// TwinCAT 3 PLC project PLC_PML
// ProgramVersion: 3.1.4023.0
// libraries:
//   PML_Base_Library, * (SPT)
//   Tc2_Math, * (Beckhoff Automation GmbH)
//   Tc2_MC2, * (Beckhoff Automation GmbH)
//   Tc2_MC2_Drive, * (Beckhoff Automation GmbH)
//   Tc2_Standard, * (Beckhoff Automation GmbH)
//   Tc2_System, * (Beckhoff Automation GmbH)
//   Tc2_Utilities, * (Beckhoff Automation GmbH)
//   Tc3_EventLogger, * (Beckhoff Automation GmbH)
//   Tc3_Module, * (Beckhoff Automation GmbH)
//   Tc3_PackML_V2, * (Beckhoff Automation GmbH)
// project tree:
//   Application/01_Application_Level_Items/02_DUT/01_ENUM/ E_PMLUnitMode.TcDUT
//   Application/01_Application_Level_Items/02_DUT/02_STRUCT/ ST_ProductionData_HMI.TcDUT
//   Application/01_Application_Level_Items/02_DUT/03_ALIAS/ T_PackMLTags.TcDUT
//   Application/01_Application_Level_Items/03_ITFs/ ITF_ProductionData.TcIO
//   Application/01_Application_Level_Items/04_HMI_Connections/ FB_MainModule_HMI_Connection.TcPOU, ST_PMLControl.TcDUT, ST_PMLControl_Simplified.TcDUT
//   Application/01_Application_Level_Items/999_VISU/ V_Application.TcVIS (not stored)
//   Application/01_Application_Level_Items/99_Templates/ FB_Module_TEMPLATE.TcPOU
//   Application/01_Application_Level_Items/ FB_ProductionMonitor.TcPOU
//   Application/02_MachineModules/ FB_TestMachine.TcPOU
//   Application/03_EquipmentModules/ FB_TestEquipment.TcPOU
//   Application/04_Components/01_Cylinder_Example/ FB_CylinderBase.TcPOU, ITF_CylinderBase.TcIO, ST_CylinderBase_HMI.TcDUT
//   Application/ MAIN.TcPOU
//   / GlobalTextList.TcGTLO (not stored), PlcTask.TcTTO (not stored), Visualization Manager.TcVMO (not stored)
// real-time tasks:
//   TASK PlcTask: cycle T#1ms, priority 20, ADS port 350
//   TASK VISU_TASK: cycle T#200000us, priority 30, ADS port 351
//   TASK Job Task: cycle default, priority 32
//   TASK MC-Task (MET): cycle T#2ms, priority 3, ADS port 521
//   TASK MC-Task (MPT): cycle T#10ms, priority 8, ADS port 531
// motion (NC):
//   TASK NC-Task 1 SAF: cycle T#2ms, priority 4, ADS port 501
//   TASK NC-Task 1 SVB: cycle T#10ms, priority 9, ADS port 511
//   AXIS Axis 1 (id 1)
//     General: UnitFlags=#x00000004
//     Dynamic: AccelerationMaximum=10000, DecelerationMaximum=10000, Acceleration=1000, Deceleration=1000, Jerk=1750
//     Velo: Maximum=1500
//     OtherSettings: AllowMotionCmdToSlave=true
//     encoder EncType=1
//       EncPara: ModuloFactor=720
//     drive DrvType=5
//       Analog: TorqueSetpointScale=10, ScaleFactorActTorque=0.1
//       TimeComp: TaskDelayCycles=1
//     controller CtrType=1
//       CtrPara: PriorControlFactor=1
//         Observer: BandWidth=20
//   AXIS Axis 2 (id 2)
//     General: UnitFlags=#x00000004
//     OtherSettings: AllowMotionCmdToSlave=true
//     encoder EncType=1
//     drive DrvType=5
//       Analog: TorqueSetpointScale=10, ScaleFactorActTorque=0.1
//       TimeComp: TaskDelayCycles=1
//     controller CtrType=1
//       CtrPara: PriorControlFactor=1
//         Observer: BandWidth=20

// ---- Application/01_Application_Level_Items/02_DUT/01_ENUM/E_PMLUnitMode.TcDUT
{attribute 'qualified_only'} //Note that this is not "Strict" since it needs to interact with the mode manager, which uses DINTs for mode
TYPE E_PMLUnitMode : (
        ePMLUnitMode_Invalid     := 0,
        ePMLUnitMode_Production  := 1,
        ePMLUnitMode_Maintenance := 2,
        ePMLUnitMode_Manual      := 3
    // User defined modes
    (*ePMLUnitMode_SemiAutomatic  :=  4,
    ePMLUnitMode_DryRun         :=  5,
	ePMLUnitMode_Standalone		:=  6,
	ePMLUnitMode_Usermode4		:=  7,
	ePMLUnitMode_Usermode5 		:=  8,
	ePMLUnitMode_Usermode6 		:=  9,
	ePMLUnitMode_Usermode7 		:=  10 *)
    ) DINT;
END_TYPE

// ---- Application/01_Application_Level_Items/02_DUT/02_STRUCT/ST_ProductionData_HMI.TcDUT
TYPE ST_ProductionData_HMI :
    STRUCT
        bHMIControlAvailable    : BOOL; //Set TRUE *FROM PLC* when HMI requests can be processed
        bIncomingHMIRequest     : BOOL; //Pulses TRUE when an HMI request is issued
        bHMICommandConfirmation : BOOL; //Confirms receipt and subsequent processing of the command sent by the HMI

        bShiftLengthHMISetRequest : BOOL;
        tShiftLengthHMISetValue   : TIME;

        bShiftProductionTargetHMISetRequest : BOOL;
        nShiftProductionTargetHMISetValue   : DINT;

        bWarningMarginHMISetRequest : BOOL;
        fWarningMarginHMISetValue   : LREAL;

        bProductionRateHMISetRequest : BOOL;
        fProductionRateHMISetValue   : LREAL;

        tShiftLength           : TIME; //Specify the time duration of a shift
        nShiftProductionTarget : DINT; //Specify the desired production count by end of shift

        nCurrentAcceptableProductionCount : DINT;
        nCurrentWarningProductionCount    : DINT;
        nCurrentShiftProductionCount      : DINT; //Number of products completed so far on the current shift
        nCurrentShiftTarget               : DINT; //Expected number of completed products at the current time in the shift
        tCurrentShiftTime                 : TIME; //Time elapsed since the start of the shift
        tRemainingShiftTime               : TIME; //Time remaining in the current shift
        tShiftStartTimeStamp              : TIMESTRUCT;
        tShiftStartTimeStamp_UTC          : STRING;
        fProductionRate_Setpoint          : LREAL;
        fProductionRate_Actual            : LREAL;
        fProductionRate_Required          : LREAL;

    END_STRUCT
END_TYPE

// ---- Application/01_Application_Level_Items/02_DUT/03_ALIAS/T_PackMLTags.TcDUT
(*	Change the type depending on the needs, minimum packml set or full
Tc3_PackML_V2.ST_PackMLv30 // Tc3_PackML_V2.ST_PackMLv30min*)
TYPE T_PackMLTags : Tc3_PackML_V2.ST_PackMLv30;
END_TYPE

// ---- Application/01_Application_Level_Items/04_HMI_Connections/ST_PMLControl.TcDUT
TYPE ST_PMLControl :
    STRUCT
        bNewCommand   : BOOL;
        bConfirmation : BOOL;

        eMode        : E_PMLUnitMode;
        eModeCommand : E_PMLUnitMode;

        eState        : E_PMLState;
        eStateCommand : E_PMLCommand;

        a_sModeNames : ARRAY[0..31] OF STRING;
    END_STRUCT
END_TYPE

// ---- Application/01_Application_Level_Items/04_HMI_Connections/ST_PMLControl_Simplified.TcDUT
TYPE ST_PMLControl_Simplified :
    STRUCT
        bConfirmation : BOOL;

        bClearEnabled : BOOL;
        bResetEnabled : BOOL;
        bStartEnabled : BOOL;
        bStopEnabled  : BOOL;

        bClearPressed : BOOL;
        bResetPressed : BOOL;
        bStartPressed : BOOL;
        bStopPressed  : BOOL;
    END_STRUCT
END_TYPE

// ---- Application/04_Components/01_Cylinder_Example/ST_CylinderBase_HMI.TcDUT
TYPE ST_CylinderBase_HMI :
    STRUCT
        //Status information
        tExtendTime     : TIME;
        tRetractTime    : TIME;
        fTimeoutFactor  : LREAL;
        bExtended       : BOOL;
        bRetracted      : BOOL;
        bExtending      : BOOL;
        bRetracting     : BOOL;
        bRetractCommand : BOOL;
        bExtendCommand  : BOOL;

        //Control information
        bHMIControlAvailable    : BOOL; //Set TRUE *FROM PLC* when HMI requests can be processed
        bIncomingHMIRequest     : BOOL; //Pulses TRUE when an HMI request is issued
        bHMICommandConfirmation : BOOL; //Confirms receipt and subsequent processing of the command sent by the HMI

        bExtendHMIRequest           : BOOL;  //HMI requests to extend the cylinder
        bRetractHMIRequest          : BOOL;  //HMI requests to retract the cylinder
        bIdleHMIRequest             : BOOL;  //HMI requests to idle the cylinder (no active output)
        bExtendTimeHMISetRequest    : BOOL;  //HMI requests to set the cylinder's expected extend time
        tExtendTimeHMISetValue      : TIME;  //HMI setpoint value for the expected extend time
        bRetractTimeHMISetRequest   : BOOL;  //HMI requests to set the cylinder's expected retract time
        tRetractTimeHMISetValue     : TIME;  //HMI setpoint value for the expected retract time
        bTimeoutFactorHMISetRequest : BOOL;  //HMI requests to set the timeout factor for the cylinder
        fTimeoutFactorHMISetValue   : LREAL; //HMI setpoint value for the cylinder's timeout factor
    END_STRUCT
END_TYPE

// ---- Application/01_Application_Level_Items/03_ITFs/ITF_ProductionData.TcIO
INTERFACE ITF_ProductionData

PROPERTY CurrentShiftAcceptableProduction : DINT
GET
END_GET
SET
END_SET
END_PROPERTY

PROPERTY CurrentShiftProductionCount : DINT
GET
END_GET
END_PROPERTY

PROPERTY CurrentShiftTarget : DINT
GET
END_GET
END_PROPERTY

PROPERTY CurrentShiftTime : TIME
GET
END_GET
END_PROPERTY

PROPERTY CurrentShiftWarningProduction : DINT
GET
END_GET
SET
END_SET
END_PROPERTY

PROPERTY NewProductionRate : bool
GET
END_GET
END_PROPERTY

PROPERTY ProductComplete : bool
GET
END_GET
SET
END_SET
END_PROPERTY

PROPERTY ProductionRate_Actual : lreal
GET
END_GET
END_PROPERTY

PROPERTY ProductionRate_Required : lreal
GET
END_GET
SET
END_SET
END_PROPERTY

PROPERTY ProductionRate_Setpoint : lreal
GET
END_GET
SET
END_SET
END_PROPERTY

PROPERTY RateAveragingCount : DINT
GET
END_GET
SET
END_SET
END_PROPERTY

PROPERTY RemainingShiftTime : TIME
GET
END_GET
SET
END_SET
END_PROPERTY

PROPERTY ShiftComplete : BOOL
GET
END_GET
END_PROPERTY

PROPERTY ShiftLength : TIME
GET
END_GET
SET
END_SET
END_PROPERTY

PROPERTY ShiftProductionTarget : DINT
GET
END_GET
SET
END_SET
END_PROPERTY

PROPERTY WarningMargin : LREAL //0 to 100, interpreted as a percentage difference between the current rate and the required rate to meet the production target, decimal values permitted
GET
END_GET
SET
END_SET
END_PROPERTY

END_INTERFACE

// ---- Application/04_Components/01_Cylinder_Example/ITF_CylinderBase.TcIO
INTERFACE ITF_CylinderBase //cylinder no feedback spring return solonoid

METHOD Extend : BOOL
END_METHOD

PROPERTY Extended : BOOL //Status bit for the position of the cylinder
GET
END_GET
END_PROPERTY

PROPERTY Extending : BOOL
GET
END_GET
END_PROPERTY

PROPERTY ExtendTime : TIME //Approximate expected time for the cylinder to complete an extension cycle
GET
END_GET
SET
END_SET
END_PROPERTY

METHOD Idle : BOOL
END_METHOD

METHOD Retract : UDINT
END_METHOD

PROPERTY Retracted : BOOL //Status bit for the position of the cylinder
GET
END_GET
END_PROPERTY

PROPERTY Retracting : BOOL
GET
END_GET
END_PROPERTY

PROPERTY RetractTime : TIME
GET
END_GET
SET
END_SET
END_PROPERTY

PROPERTY TimeoutFactor : LREAL //Multiplicative factor that determines error timeout threshold based on the expected time
GET
END_GET
SET
END_SET
END_PROPERTY

END_INTERFACE

// ---- Application/01_Application_Level_Items/04_HMI_Connections/FB_MainModule_HMI_Connection.TcPOU
FUNCTION_BLOCK FB_MainModule_HMI_Connection
VAR CONSTANT
    //Constant declarations
    PRODUCTION_DATA_ALARM_COUNT : UDINT := 16;
END_VAR
VAR PERSISTENT
    //ITF_ProductionData internal variables
    tShiftLength             : TIME  := T#10M;
    nShiftProductionTarget   : DINT  := 1000;
    fWarningMargin           : LREAL := 10;
    fProductionRate_Setpoint : LREAL := 30;
    nRateAveragingCount      : DINT  := 10;
END_VAR
VAR
    //Internal Property Variables
    itfMainModule : ITF_PMLModuleBase;

    //Program Tree variables
    fbModuleTree         : FB_Tree_IndexBased;
    a_stMachineTreeNodes : ARRAY[0..63] OF ST_Tree_IndexBased_Node;
    sTopLevelMachine     : STRING;

    //PML Control Variables
    stMainPMLControl_Simplified : ST_PMLControl_Simplified;
    stMainPMLControl_Standard   : ST_PMLControl;

    //Status Variables
    stMainProductionData : REFERENCE TO ST_ProductionData_HMI;

    //Production Data variables
    bShiftComplete                    : BOOL;
    bProductComplete                  : BOOL;
    nCurrentShiftProductionCount      : INT;
    nCurrentShiftTarget               : DINT;
    tCurrentShiftTime                 : TIME;
    tRemainingShiftTime               : TIME;
    tShiftStartTimeStamp              : TIMESTRUCT;
    tShiftStartTimeStamp_UTC          : STRING;
    nCurrentWarningProductionCount    : DINT;
    nCurrentAcceptableProductionCount : DINT;

    fProductionRate_Required : LREAL;
    fProductionRate_Actual   : LREAL;

    a_nLastProductTimestamps : ARRAY[1..100] OF ULINT; //Array of ULINT values (1 unit = 1ns) for the relative time of each of the last 100 completed products
    fbShiftTimer             : TON;
    fbGetTime                : NT_GetTime;
    fbProductComplete_RT     : R_TRIG;

    bResetMaxProductionCount   : BOOL;
    bResetTotalProductionCount : BOOL;

    nMaxProductionCount   : DINT;
    nTotalProductionCount : DINT;

    stProductionDataHMI      : ST_ProductionData_HMI;
    fbFIFO                   : FB_FIFO_ULINT_Array;
    a_fbProductionDataAlarms : ARRAY[1..PRODUCTION_DATA_ALARM_COUNT] OF FB_TcAlarm;
    fTemp                    : LREAL;

    //Other Internal Variables
    bInitialized : BOOL;
    i            : UDINT;

END_VAR

METHOD CyclicLogic : BOOL
VAR_INPUT
END_VAR
IF NOT bInitialized THEN
    initialize();
    bInitialized := TRUE;
END_IF

stMainPMLControl_Standard.eMode  := itfMainModule.Mode;
stMainPMLControl_Standard.eState := itfMainModule.State;

FOR i := 1 TO 5 DO
    stMainPMLControl_Standard.a_sModeNames[i] := F_UnitModeToString(i);
	
END_FOR

stMainPMLControl_Standard.eState := itfMainModule.State;
stMainPMLControl_Standard.eMode  := itfMainModule.Mode;

MainCycleControl();

//bProductComplete := itfMainModule.ProductComplete;

ProductionMonitor();
HMICommunication();

//itfMainModule.ProductionRate_Setpoint := fProductionRate_Setpoint;
END_METHOD

PROPERTY DataStructure_Adder : ITF_Tree_IndexBased
GET
DataStructure_Adder := fbModuleTree;
END_GET
END_PROPERTY

METHOD HMICommunication : BOOL
VAR_INPUT
END_VAR
//Production Data================================================================================================================================================

//Process HMI requests
IF stProductionDataHMI.bIncomingHMIRequest AND NOT stProductionDataHMI.bHMICommandConfirmation
    THEN //If a request has been issued by the HMI, and a previous request has not just E_SequenceState.Finished being processed
    IF stProductionDataHMI.bShiftProductionTargetHMISetRequest THEN
        nShiftProductionTarget                      := stProductionDataHMI.nShiftProductionTargetHMISetValue;
        stProductionDataHMI.bHMICommandConfirmation := TRUE; //Confirm that the request has been processed
    END_IF

    IF stProductionDataHMI.bWarningMarginHMISetRequest THEN
        fWarningMargin                              := stProductionDataHMI.fWarningMarginHMISetValue;
        stProductionDataHMI.bHMICommandConfirmation := TRUE; //Confirm that the request has been processed
    END_IF

    IF stProductionDataHMI.bShiftLengthHMISetRequest THEN
        tShiftLength                                := stProductionDataHMI.tShiftLengthHMISetValue;
        stProductionDataHMI.bHMICommandConfirmation := TRUE; //Confirm that the request has been processed
    END_IF

    IF stProductionDataHMI.bProductionRateHMISetRequest THEN
        fProductionRate_Setpoint                    := stProductionDataHMI.fProductionRateHMISetValue;
        stProductionDataHMI.bHMICommandConfirmation := TRUE; //Confirm that the request has been processed
    END_IF
END_IF

//Update HMI Status Info
stProductionDataHMI.tShiftLength                      := tShiftLength;
stProductionDataHMI.nShiftProductionTarget            := nShiftProductionTarget;
stProductionDataHMI.nCurrentShiftProductionCount      := nCurrentShiftProductionCount;
stProductionDataHMI.nCurrentShiftTarget               := nCurrentShiftTarget;
stProductionDataHMI.nCurrentAcceptableProductionCount := nCurrentAcceptableProductionCount;
stProductionDataHMI.nCurrentWarningProductionCount    := nCurrentWarningProductionCount;
stProductionDataHMI.tCurrentShiftTime                 := tCurrentShiftTime;
stProductionDataHMI.tRemainingShiftTime               := tRemainingShiftTime;
stProductionDataHMI.tShiftStartTimeStamp              := tShiftStartTimeStamp;
stProductionDataHMI.tShiftStartTimeStamp_UTC          := tShiftStartTimeStamp_UTC;
stProductionDataHMI.fProductionRate_Setpoint          := F_LREAL_RoundToPlace(fProductionRate_Setpoint, 1);
stProductionDataHMI.fProductionRate_Actual            := F_LREAL_RoundToPlace(fProductionRate_Actual, 1);
stProductionDataHMI.fProductionRate_Required          := F_LREAL_RoundToPlace(fProductionRate_Required, 1);
END_METHOD

METHOD initialize : BOOL
VAR_INPUT
END_VAR
sTopLevelMachine := itfMainModule.ModuleName;

fbModuleTree(a_stNodes := a_stMachineTreeNodes, sHead := sTopLevelMachine);

F_CreateAllEventsInClass(p_aAlarms  := a_fbProductionDataAlarms,
                         nClassSize := SIZEOF(TC_EVENTS.ProductionData),
                         pInitEvent := ADR(TC_EVENTS.ProductionData.InitReferenceEvent),
                         sPrefix    := MainModule.ModuleName);
END_METHOD

METHOD MainCycleControl : BOOL
VAR_INPUT
END_VAR
//Simplified Commands
//Handle button presses
IF NOT stMainPMLControl_Simplified.bConfirmation AND stMainPMLControl_Simplified.bStartPressed THEN
    IF stMainPMLControl_Standard.eState = Tc3_PackML_V2.E_PMLState.ePMLState_Idle THEN
        itfMainModule.StateCommand := Tc3_PackML_V2.E_PMLCommand.ePMLCommand_Start;
    ELSIF stMainPMLControl_Standard.eState = Tc3_PackML_V2.E_PMLState.ePMLState_Held THEN
        itfMainModule.StateCommand := Tc3_PackML_V2.E_PMLCommand.ePMLCommand_Unhold;
    END_IF

    stMainPMLControl_Simplified.bConfirmation := TRUE;
END_IF

IF NOT stMainPMLControl_Simplified.bConfirmation AND stMainPMLControl_Simplified.bStopPressed THEN
    itfMainModule.StateCommand                := Tc3_PackML_V2.E_PMLCommand.ePMLCommand_Stop;
    stMainPMLControl_Simplified.bConfirmation := TRUE;
END_IF

IF NOT stMainPMLControl_Simplified.bConfirmation AND stMainPMLControl_Simplified.bResetPressed THEN
    itfMainModule.StateCommand                := Tc3_PackML_V2.E_PMLCommand.ePMLCommand_Reset;
    stMainPMLControl_Simplified.bConfirmation := TRUE;
END_IF

IF NOT stMainPMLControl_Simplified.bConfirmation AND stMainPMLControl_Simplified.bClearPressed THEN
    itfMainModule.StateCommand                := Tc3_PackML_V2.E_PMLCommand.ePMLCommand_Clear;
    stMainPMLControl_Simplified.bConfirmation := TRUE;
END_IF

//Handle enabling of the Start button
IF stMainPMLControl_Standard.eState = Tc3_PackML_V2.E_PMLState.ePMLState_Idle
       OR stMainPMLControl_Standard.eState = Tc3_PackML_V2.E_PMLState.ePMLState_Held THEN
    stMainPMLControl_Simplified.bStartEnabled := TRUE;
ELSE
    stMainPMLControl_Simplified.bStartEnabled := FALSE;
END_IF

//Handle enabling of the Stop button
IF stMainPMLControl_Standard.eState <> Tc3_PackML_V2.E_PMLState.ePMLState_Stopped
       AND stMainPMLControl_Standard.eState <> Tc3_PackML_V2.E_PMLState.ePMLState_Clearing
       AND stMainPMLControl_Standard.eState <> Tc3_PackML_V2.E_PMLState.ePMLState_Aborted
       AND stMainPMLControl_Standard.eState <> Tc3_PackML_V2.E_PMLState.ePMLState_Aborting
       AND stMainPMLControl_Standard.eState <> Tc3_PackML_V2.E_PMLState.ePMLState_Undefined THEN
    stMainPMLControl_Simplified.bStopEnabled := TRUE;
ELSE
    stMainPMLControl_Simplified.bStopEnabled := FALSE;
END_IF

//Handle enabling of the Reset button
IF stMainPMLControl_Standard.eState = Tc3_PackML_V2.E_PMLState.ePMLState_Complete
       OR stMainPMLControl_Standard.eState = Tc3_PackML_V2.E_PMLState.ePMLState_Stopped THEN
    stMainPMLControl_Simplified.bResetEnabled := TRUE;
ELSE
    stMainPMLControl_Simplified.bResetEnabled := FALSE;
END_IF

//Handle enabling of the Clear button
IF stMainPMLControl_Standard.eState = Tc3_PackML_V2.E_PMLState.ePMLState_Aborted THEN
    stMainPMLControl_Simplified.bClearEnabled := TRUE;
ELSE
    stMainPMLControl_Simplified.bClearEnabled := FALSE;
END_IF

//Standard Commands

IF NOT stMainPMLControl_Standard.bConfirmation AND stMainPMLControl_Standard.bNewCommand THEN
    IF stMainPMLControl_Standard.eStateCommand <> E_PMLCommand.ePMLCommand_Undefined THEN
        itfMainModule.StateCommand              := stMainPMLControl_Standard.eStateCommand;
        stMainPMLControl_Standard.bConfirmation := TRUE;
    END_IF

    IF stMainPMLControl_Standard.eModeCommand <> E_PMLUnitMode.ePMLUnitMode_Invalid THEN
        itfMainModule.StateCommand              := stMainPMLControl_Standard.eStateCommand;
        stMainPMLControl_Standard.bConfirmation := TRUE;
    END_IF
END_IF
END_METHOD

PROPERTY MainModule : ITF_PMLModuleBase
GET
MainModule := itfMainModule;
END_GET
SET
itfMainModule := MainModule;
END_SET
END_PROPERTY

METHOD ProductionMonitor : BOOL
VAR_INPUT
END_VAR
IF NOT bInitialized THEN
    initialize();
    bInitialized := TRUE;
END_IF

fbGetTime(NETID   := '',
          START   := NOT bShiftComplete,
          TMOUT   :=,
          BUSY    =>,
          ERR     =>,
          ERRID   =>,
          TIMESTR => tShiftStartTimeStamp);

IF NOT fbGetTime.BUSY THEN
    tShiftStartTimeStamp_UTC := SYSTEMTIME_TO_ISO8601(tShiftstartTimeStamp, 0, FALSE, 3);
    tShiftStartTimeStamp_UTC := LEFT(STR := tShiftStartTimeStamp_UTC, SIZE := FIND(tShiftStartTimeStamp_UTC, '+') - 1);
END_IF

fbFIFO(a_FIFO := a_nLastProductTimestamps);

fbShiftTimer(IN := NOT bShiftComplete, PT := tShiftLength, Q => bShiftComplete, ET => tCurrentShiftTime);
tRemainingShiftTime := tShiftLength - tCurrentShiftTime;

IF TIME_TO_DINT(tRemainingShiftTime) > 0 THEN
    fProductionRate_Required :=
        DINT_TO_LREAL(nShiftProductionTarget - nCurrentShiftProductionCount) / (TIME_TO_LREAL(tRemainingShiftTime) / 1000 / 60);

    nCurrentAcceptableProductionCount := nCurrentShiftTarget;

    nCurrentWarningProductionCount :=
        nShiftProductionTarget
            - (LREAL_TO_DINT((fProductionRate_Actual * (1 + fWarningMargin / 100)) * (TIME_TO_LREAL(tRemainingShiftTime) / 1000 / 60)));

    IF nCurrentWarningProductionCount < 0 THEN
        nCurrentWarningProductionCount := 0;
    END_IF
END_IF

fbProductComplete_RT(CLK := bProductComplete);

IF fbProductComplete_RT.Q THEN
    nCurrentShiftProductionCount := nCurrentShiftProductionCount + 1;
    nTotalProductionCount        := nTotalProductionCount + 1;

    IF nCurrentShiftProductionCount > nMaxProductionCount THEN
        nMaxProductionCount := nCurrentShiftProductionCount;
    END_IF

    fbFIFO.AddEntry(nEntry := F_GetSystemTime());
END_IF

IF (fbFIFO.EntryCount > nRateAveragingCount) THEN
    fbFIFO.RemoveEntry();
END_IF

fTemp := (TIME_TO_LREAL(ULINT_TO_TIME(fbFIFO.LastInValue - fbFIFO.NextOutValue)) / 10000 / 1000 / 60);

IF fTemp > 0 AND fbFIFO.EntryCount > 1 THEN
    fProductionRate_Actual := F_LREAL_RoundToPlace(DINT_TO_LREAL(fbFIFO.EntryCount - 1) / fTemp, 2);
END_IF

IF TIME_TO_DINT(tShiftLength) > 0 THEN
    nCurrentShiftTarget := LREAL_TO_DINT((TIME_TO_LREAL(tCurrentShiftTime) / TIME_TO_LREAL(tShiftLength)) * DINT_TO_LREAL(nShiftProductionTarget));
END_IF

IF bShiftComplete THEN
    nCurrentShiftProductionCount := 0;
END_IF

IF bResetMaxProductionCount THEN
    nMaxProductionCount := nCurrentShiftProductionCount;
END_IF

IF bResetTotalProductionCount THEN
    nTotalProductionCount := 0;
END_IF
END_METHOD

END_FUNCTION_BLOCK

// ---- Application/01_Application_Level_Items/99_Templates/FB_Module_TEMPLATE.TcPOU
FUNCTION_BLOCK FB_Module_TEMPLATE EXTENDS FB_PMLModuleBase
VAR
    //Define the Sub modules here for this module. (If any)  Also set the Interfaces in the initialize method.
    (*fbSubModule1				: FB_ApplicationModule_TEMPLATE := (ModuleName :=  'Test Module 1');
	*)
    (*fbSubModule2				: FB_ApplicationModule_TEMPLATE := (ModuleName :=  'Test Module 2');
	*)
    //temporary array of module base interfaces to be copied over to the base class a_itfPackMLBase variable
    a_ITF_PackMLBase_init : ARRAY[1..MAX_NO_OF_SUBMODULES] OF ITF_PMLModuleBase
        := [ (*	fbSubModule1,
																							 	fbSubModule2*) ];

    //Define the components here for this module. (If any) Also set the Interfaces in the initialize method.
    (*fbComponent1				: FB_ComponentBase (Extension):= (Name := 'Test Component 1');
	*)
    (*fbComponent2				: FB_ComponentBase (Extension):= (Name := 'Test Component 2');
	*)
    //temporary array of module base interfaces to be copied over to the base class a_itfPackMLBase variable
    a_ITF_Components_init : ARRAY[1..GVL_PML_Base.MAX_NO_OF_COMPONENTS] OF ITF_ComponentBase := [ (*	fbComponent1,
																											fbComponent2*)
    ];

END_VAR

//*********************************************************
//Body of block is not called by base code, only implement application
//code in CyclicUpdate or in methods called by it or its subcalls
//*********************************************************

METHOD Aborted
CASE eMode OF
    //	====================================================================PRODUCTION MODE=========================================================	
    E_PMLUnitMode.ePMLUnitMode_Production:
        ;
    //	====================================================================MANUAL MODE=============================================================	
    E_PMLUnitMode.ePMLUnitMode_Manual:
        ;
    //	=====================================================================MAINTENANCE MODE=======================================================	
    E_PMLUnitMode.ePMLUnitMode_Maintenance:
        ;
    //	=====================================================================CUSTOM MODE 1==========================================================	
    (*	E_PMLUnitMode.ePMLUnitMode_YOURCUSTOMMODE		
		;*)
    //	======================================================================INVALID MODE==========================================================	
    E_PMLUnitMode.ePMLUnitMode_Invalid:
        ;
END_CASE
END_METHOD

METHOD Aborting
//bNoStateTasksToComplete := TRUE;		// Change to False if not used

//Implement state Tasks here
(*
IF (insert your completion conditions) THEN

bStateTasksComplete := TRUE;				//Once these actions are completed successfully, set bStateTasksComplete to allow the base code to advance once all children have also reached the proper state

END_IF
*)

SUPER^.Aborting();

(*	Reference State Machine for mode specific actions - Be sure to paste above the SUPER^ Call if used - Delete if not needed

CASE eMode OF
//	====================================================================PRODUCTION MODE=========================================================	
	E_PMLUnitMode.ePMLUnitMode_Production:			
		;
//	====================================================================MANUAL MODE=============================================================	
	E_PMLUnitMode.ePMLUnitMode_Manual:				
		;
//	=====================================================================MAINTENANCE MODE=======================================================	
	E_PMLUnitMode.ePMLUnitMode_Maintenance:			
		;	
//	=====================================================================CUSTOM MODE 1==========================================================	
(*	E_PMLUnitMode.ePMLUnitMode_YOURCUSTOMMODE		
		;*)
//	======================================================================INVALID MODE==========================================================	
	E_PMLUnitMode.ePMLUnitMode_Invalid:				
		;
END_CASE
*)
END_METHOD

METHOD Clearing
//bNoStateTasksToComplete := TRUE;		// Change to False if not used

//Implement state Tasks here
(*
IF (insert your completion conditions) THEN

bStateTasksComplete := TRUE;				//Once these actions are completed successfully, set bStateTasksComplete to allow the base code to advance once all children have also reached the proper state

END_IF
*)

SUPER^.Clearing();
(*	Reference State Machine for mode specific actions - Be sure to paste above the SUPER^ Call if used - Delete if not needed

CASE eMode OF
//	====================================================================PRODUCTION MODE=========================================================	
	E_PMLUnitMode.ePMLUnitMode_Production:			
		;
//	====================================================================MANUAL MODE=============================================================	
	E_PMLUnitMode.ePMLUnitMode_Manual:				
		;
//	=====================================================================MAINTENANCE MODE=======================================================	
	E_PMLUnitMode.ePMLUnitMode_Maintenance:			
		;	
//	=====================================================================CUSTOM MODE 1==========================================================	
(*	E_PMLUnitMode.ePMLUnitMode_YOURCUSTOMMODE		
		;*)
//	======================================================================INVALID MODE==========================================================	
	E_PMLUnitMode.ePMLUnitMode_Invalid:				
		;
END_CASE
*)
END_METHOD

METHOD Complete
CASE eMode OF
    //	====================================================================PRODUCTION MODE=========================================================	
    E_PMLUnitMode.ePMLUnitMode_Production:
        ;
    //	====================================================================MANUAL MODE=============================================================	
    E_PMLUnitMode.ePMLUnitMode_Manual:
        ;
    //	=====================================================================MAINTENANCE MODE=======================================================	
    E_PMLUnitMode.ePMLUnitMode_Maintenance:
        ;
    //	=====================================================================CUSTOM MODE 1==========================================================	
    (*	E_PMLUnitMode.ePMLUnitMode_YOURCUSTOMMODE		
		;*)
    //	======================================================================INVALID MODE==========================================================	
    E_PMLUnitMode.ePMLUnitMode_Invalid:
        ;
END_CASE
END_METHOD

METHOD Completing
//bNoStateTasksToComplete := TRUE;		// Change to False if not used

//Implement state Tasks here
(*
IF (insert your completion conditions) THEN

bStateTasksComplete := TRUE;				//Once these actions are completed successfully, set bStateTasksComplete to allow the base code to advance once all children have also reached the proper state

END_IF
*)

SUPER^.Completing();

(*	Reference State Machine for mode specific actions - Be sure to paste above the SUPER^ Call if used - Delete if not needed

CASE eMode OF
//	====================================================================PRODUCTION MODE=========================================================	
	E_PMLUnitMode.ePMLUnitMode_Production:			
		;
//	====================================================================MANUAL MODE=============================================================	
	E_PMLUnitMode.ePMLUnitMode_Manual:				
		;
//	=====================================================================MAINTENANCE MODE=======================================================	
	E_PMLUnitMode.ePMLUnitMode_Maintenance:			
		;	
//	=====================================================================CUSTOM MODE 1==========================================================	
(*	E_PMLUnitMode.ePMLUnitMode_YOURCUSTOMMODE		
		;*)
//	======================================================================INVALID MODE==========================================================	
	E_PMLUnitMode.ePMLUnitMode_Invalid:				
		;
END_CASE
*)
END_METHOD

// 
// Cyclic Code
METHOD CyclicLogic
VAR
    i : UDINT; //Generic iteration value
END_VAR
// Main loop of the parent module
SUPER^.CyclicLogic();
END_METHOD

METHOD Execute
CASE eMode OF
    //	====================================================================PRODUCTION MODE=========================================================	
    E_PMLUnitMode.ePMLUnitMode_Production:
        ;
    //	====================================================================MANUAL MODE=============================================================	
    E_PMLUnitMode.ePMLUnitMode_Manual:
        ;
    //	=====================================================================MAINTENANCE MODE=======================================================	
    E_PMLUnitMode.ePMLUnitMode_Maintenance:
        ;
    //	=====================================================================CUSTOM MODE 1==========================================================	
    (*	E_PMLUnitMode.ePMLUnitMode_YOURCUSTOMMODE		
		;*)
    //	======================================================================INVALID MODE==========================================================	
    E_PMLUnitMode.ePMLUnitMode_Invalid:
        ;
END_CASE
END_METHOD

METHOD Held
CASE eMode OF
    //	====================================================================PRODUCTION MODE=========================================================	
    E_PMLUnitMode.ePMLUnitMode_Production:
        ;
    //	====================================================================MANUAL MODE=============================================================	
    E_PMLUnitMode.ePMLUnitMode_Manual:
        ;
    //	=====================================================================MAINTENANCE MODE=======================================================	
    E_PMLUnitMode.ePMLUnitMode_Maintenance:
        ;
    //	=====================================================================CUSTOM MODE 1==========================================================	
    (*	E_PMLUnitMode.ePMLUnitMode_YOURCUSTOMMODE		
		;*)
    //	======================================================================INVALID MODE==========================================================	
    E_PMLUnitMode.ePMLUnitMode_Invalid:
        ;
END_CASE
END_METHOD

METHOD Holding
//bNoStateTasksToComplete := TRUE;		// Change to False if not used

//Implement state Tasks here
(*
IF (insert your completion conditions) THEN

bStateTasksComplete := TRUE;				//Once these actions are completed successfully, set bStateTasksComplete to allow the base code to advance once all children have also reached the proper state

END_IF
*)

SUPER^.Holding();

(*	Reference State Machine for mode specific actions - Be sure to paste above the SUPER^ Call if used - Delete if not needed

CASE eMode OF
//	====================================================================PRODUCTION MODE=========================================================	
	E_PMLUnitMode.ePMLUnitMode_Production:			
		;
//	====================================================================MANUAL MODE=============================================================	
	E_PMLUnitMode.ePMLUnitMode_Manual:				
		;
//	=====================================================================MAINTENANCE MODE=======================================================	
	E_PMLUnitMode.ePMLUnitMode_Maintenance:			
		;	
//	=====================================================================CUSTOM MODE 1==========================================================	
(*	E_PMLUnitMode.ePMLUnitMode_YOURCUSTOMMODE		
		;*)
//	======================================================================INVALID MODE==========================================================	
	E_PMLUnitMode.ePMLUnitMode_Invalid:				
		;
END_CASE
*)
END_METHOD

METHOD Idle
CASE eMode OF
    //	====================================================================PRODUCTION MODE=========================================================	
    E_PMLUnitMode.ePMLUnitMode_Production:
        ;
    //	====================================================================MANUAL MODE=============================================================	
    E_PMLUnitMode.ePMLUnitMode_Manual:
        ;
    //	=====================================================================MAINTENANCE MODE=======================================================	
    E_PMLUnitMode.ePMLUnitMode_Maintenance:
        ;
    //	=====================================================================CUSTOM MODE 1==========================================================	
    (*	E_PMLUnitMode.ePMLUnitMode_YOURCUSTOMMODE		
		;*)
    //	======================================================================INVALID MODE==========================================================	
    E_PMLUnitMode.ePMLUnitMode_Invalid:
        ;
END_CASE
END_METHOD

METHOD Initialize
VAR
    i : UDINT; //Generic iteration value
END_VAR
// Define the interfaces to the different subunits (Must take place before SUPER^.initialize call)
FOR i := 1 TO MAX_NO_OF_SUBMODULES DO
    a_ITF_PackMLBase[i] := a_ITF_PackMLBase_init[i];
END_FOR

FOR i := 1 TO MAX_NO_OF_COMPONENTS DO
    a_ITF_Components[i] := a_ITF_Components_init[i];
END_FOR

// Init of the parent class object (Must be called AFTER most local init code, since the sub module interface array assignments should be made here, and then operated on within the module base init
SUPER^.Initialize();
END_METHOD

METHOD Resetting
//bNoStateTasksToComplete := TRUE;		// Change to False if not used

//Implement state Tasks here
(*
IF (insert your completion conditions) THEN

bStateTasksComplete := TRUE;				//Once these actions are completed successfully, set bStateTasksComplete to allow the base code to advance once all children have also reached the proper state

END_IF
*)

SUPER^.Resetting();

(*	Reference State Machine for mode specific actions - Be sure to paste above the SUPER^ Call if used - Delete if not needed

CASE eMode OF
//	====================================================================PRODUCTION MODE=========================================================	
	E_PMLUnitMode.ePMLUnitMode_Production:			
		;
//	====================================================================MANUAL MODE=============================================================	
	E_PMLUnitMode.ePMLUnitMode_Manual:				
		;
//	=====================================================================MAINTENANCE MODE=======================================================	
	E_PMLUnitMode.ePMLUnitMode_Maintenance:			
		;	
//	=====================================================================CUSTOM MODE 1==========================================================	
(*	E_PMLUnitMode.ePMLUnitMode_YOURCUSTOMMODE		
		;*)
//	======================================================================INVALID MODE==========================================================	
	E_PMLUnitMode.ePMLUnitMode_Invalid:				
		;
END_CASE
*)
END_METHOD

METHOD Starting
//bNoStateTasksToComplete := TRUE;		// Change to False if not used

//Implement state Tasks here
(*
IF (insert your completion conditions) THEN

bStateTasksComplete := TRUE;				//Once these actions are completed successfully, set bStateTasksComplete to allow the base code to advance once all children have also reached the proper state

END_IF
*)

SUPER^.Starting();

(*	Reference State Machine for mode specific actions - Be sure to paste above the SUPER^ Call if used - Delete if not needed

CASE eMode OF
//	====================================================================PRODUCTION MODE=========================================================	
	E_PMLUnitMode.ePMLUnitMode_Production:			
		;
//	====================================================================MANUAL MODE=============================================================	
	E_PMLUnitMode.ePMLUnitMode_Manual:				
		;
//	=====================================================================MAINTENANCE MODE=======================================================	
	E_PMLUnitMode.ePMLUnitMode_Maintenance:			
		;	
//	=====================================================================CUSTOM MODE 1==========================================================	
(*	E_PMLUnitMode.ePMLUnitMode_YOURCUSTOMMODE		
		;*)
//	======================================================================INVALID MODE==========================================================	
	E_PMLUnitMode.ePMLUnitMode_Invalid:				
		;
END_CASE
*)
END_METHOD

METHOD Stopped
CASE eMode OF
    //	====================================================================PRODUCTION MODE=========================================================	
    E_PMLUnitMode.ePMLUnitMode_Production:
        ;
    //	====================================================================MANUAL MODE=============================================================	
    E_PMLUnitMode.ePMLUnitMode_Manual:
        ;
    //	=====================================================================MAINTENANCE MODE=======================================================	
    E_PMLUnitMode.ePMLUnitMode_Maintenance:
        ;
    //	=====================================================================CUSTOM MODE 1==========================================================	
    (*	E_PMLUnitMode.ePMLUnitMode_YOURCUSTOMMODE		
		;*)
    //	======================================================================INVALID MODE==========================================================	
    E_PMLUnitMode.ePMLUnitMode_Invalid:
        ;
END_CASE
END_METHOD

METHOD Stopping
//bNoStateTasksToComplete := TRUE;		// Change to False if not used

//Implement state Tasks here
(*
IF (insert your completion conditions) THEN

bStateTasksComplete := TRUE;				//Once these actions are completed successfully, set bStateTasksComplete to allow the base code to advance once all children have also reached the proper state

END_IF
*)

SUPER^.Stopping();

(*	Reference State Machine for mode specific actions - Be sure to paste above the SUPER^ Call if used - Delete if not needed

CASE eMode OF
//	====================================================================PRODUCTION MODE=========================================================	
	E_PMLUnitMode.ePMLUnitMode_Production:			
		;
//	====================================================================MANUAL MODE=============================================================	
	E_PMLUnitMode.ePMLUnitMode_Manual:				
		;
//	=====================================================================MAINTENANCE MODE=======================================================	
	E_PMLUnitMode.ePMLUnitMode_Maintenance:			
		;	
//	=====================================================================CUSTOM MODE 1==========================================================	
(*	E_PMLUnitMode.ePMLUnitMode_YOURCUSTOMMODE		
		;*)
//	======================================================================INVALID MODE==========================================================	
	E_PMLUnitMode.ePMLUnitMode_Invalid:				
		;
END_CASE
*)
END_METHOD

METHOD Suspended
CASE eMode OF
    //	====================================================================PRODUCTION MODE=========================================================	
    E_PMLUnitMode.ePMLUnitMode_Production:
        ;
    //	====================================================================MANUAL MODE=============================================================	
    E_PMLUnitMode.ePMLUnitMode_Manual:
        ;
    //	=====================================================================MAINTENANCE MODE=======================================================	
    E_PMLUnitMode.ePMLUnitMode_Maintenance:
        ;
    //	=====================================================================CUSTOM MODE 1==========================================================	
    (*	E_PMLUnitMode.ePMLUnitMode_YOURCUSTOMMODE		
		;*)
    //	======================================================================INVALID MODE==========================================================	
    E_PMLUnitMode.ePMLUnitMode_Invalid:
        ;
END_CASE
END_METHOD

METHOD Suspending
//bNoStateTasksToComplete := TRUE;		// Change to False if not used

//Implement state Tasks here
(*
IF (insert your completion conditions) THEN

bStateTasksComplete := TRUE;				//Once these actions are completed successfully, set bStateTasksComplete to allow the base code to advance once all children have also reached the proper state

END_IF
*)

SUPER^.Suspending();

(*	Reference State Machine for mode specific actions - Be sure to paste above the SUPER^ Call if used - Delete if not needed

CASE eMode OF
//	====================================================================PRODUCTION MODE=========================================================	
	E_PMLUnitMode.ePMLUnitMode_Production:			
		;
//	====================================================================MANUAL MODE=============================================================	
	E_PMLUnitMode.ePMLUnitMode_Manual:				
		;
//	=====================================================================MAINTENANCE MODE=======================================================	
	E_PMLUnitMode.ePMLUnitMode_Maintenance:			
		;	
//	=====================================================================CUSTOM MODE 1==========================================================	
(*	E_PMLUnitMode.ePMLUnitMode_YOURCUSTOMMODE		
		;*)
//	======================================================================INVALID MODE==========================================================	
	E_PMLUnitMode.ePMLUnitMode_Invalid:				
		;
END_CASE
*)
END_METHOD

METHOD Undefined
CASE eMode OF
    //	====================================================================PRODUCTION MODE=========================================================	
    E_PMLUnitMode.ePMLUnitMode_Production:
        ;
    //	====================================================================MANUAL MODE=============================================================	
    E_PMLUnitMode.ePMLUnitMode_Manual:
        ;
    //	=====================================================================MAINTENANCE MODE=======================================================	
    E_PMLUnitMode.ePMLUnitMode_Maintenance:
        ;
    //	=====================================================================CUSTOM MODE 1==========================================================	
    (*	E_PMLUnitMode.ePMLUnitMode_YOURCUSTOMMODE		
		;*)
    //	======================================================================INVALID MODE==========================================================	
    E_PMLUnitMode.ePMLUnitMode_Invalid:
        ;
END_CASE
END_METHOD

METHOD Unholding
//bNoStateTasksToComplete := TRUE;		// Change to False if not used

//Implement state Tasks here
(*
IF (insert your completion conditions) THEN

bStateTasksComplete := TRUE;				//Once these actions are completed successfully, set bStateTasksComplete to allow the base code to advance once all children have also reached the proper state

END_IF
*)

SUPER^.Unholding();

(*	Reference State Machine for mode specific actions - Be sure to paste above the SUPER^ Call if used - Delete if not needed

CASE eMode OF
//	====================================================================PRODUCTION MODE=========================================================	
	E_PMLUnitMode.ePMLUnitMode_Production:			
		;
//	====================================================================MANUAL MODE=============================================================	
	E_PMLUnitMode.ePMLUnitMode_Manual:				
		;
//	=====================================================================MAINTENANCE MODE=======================================================	
	E_PMLUnitMode.ePMLUnitMode_Maintenance:			
		;	
//	=====================================================================CUSTOM MODE 1==========================================================	
(*	E_PMLUnitMode.ePMLUnitMode_YOURCUSTOMMODE		
		;*)
//	======================================================================INVALID MODE==========================================================	
	E_PMLUnitMode.ePMLUnitMode_Invalid:				
		;
END_CASE
*)
END_METHOD

METHOD Unsuspending
//bNoStateTasksToComplete := TRUE;		// Change to False if not used

//Implement state Tasks here
(*
IF (insert your completion conditions) THEN

bStateTasksComplete := TRUE;				//Once these actions are completed successfully, set bStateTasksComplete to allow the base code to advance once all children have also reached the proper state

END_IF
*)

SUPER^.Unsuspending();

(*	Reference State Machine for mode specific actions - Be sure to paste above the SUPER^ Call if used - Delete if not needed

CASE eMode OF
//	====================================================================PRODUCTION MODE=========================================================	
	E_PMLUnitMode.ePMLUnitMode_Production:			
		;
//	====================================================================MANUAL MODE=============================================================	
	E_PMLUnitMode.ePMLUnitMode_Manual:				
		;
//	=====================================================================MAINTENANCE MODE=======================================================	
	E_PMLUnitMode.ePMLUnitMode_Maintenance:			
		;	
//	=====================================================================CUSTOM MODE 1==========================================================	
(*	E_PMLUnitMode.ePMLUnitMode_YOURCUSTOMMODE		
		;*)
//	======================================================================INVALID MODE==========================================================	
	E_PMLUnitMode.ePMLUnitMode_Invalid:				
		;
END_CASE
*)
END_METHOD

END_FUNCTION_BLOCK

// ---- Application/01_Application_Level_Items/FB_ProductionMonitor.TcPOU
FUNCTION_BLOCK FB_ProductionMonitor IMPLEMENTS ITF_ProductionData
VAR CONSTANT
    //Constant declarations
    PRODUCTION_DATA_ALARM_COUNT : UDINT := 16;
END_VAR
VAR PERSISTENT
    //ITF_ProductionData internal variables
    tShiftLength             : TIME  := T#10M;
    nShiftProductionTarget   : DINT  := 1000;
    fWarningMargin           : LREAL := 10;
    fProductionRate_Setpoint : LREAL := 30;
    nRateAveragingCount      : DINT  := 10;
END_VAR
VAR
    //ITF_ProductionData internal variables + Other Production related variables
    bShiftComplete                    : BOOL;
    bProductComplete                  : BOOL;
    nCurrentShiftProductionCount      : INT;
    nCurrentShiftTarget               : DINT;
    tCurrentShiftTime                 : TIME;
    tRemainingShiftTime               : TIME;
    nCurrentWarningProductionCount    : DINT;
    nCurrentAcceptableProductionCount : DINT;

    fProductionRate_Required : LREAL;
    fProductionRate_Actual   : LREAL;

    a_nLastProductTimestamps  : ARRAY[1..100] OF ULINT; //Array of ULINT values (1 unit = 1ns) for the relative time of each of the last 100 completed products
    fbShiftTimer              : TON;
    fbProductComplete_RT      : R_TRIG;
    bNewProductionRate        : BOOL;
    fLastTargetProductionRate : LREAL;

    bResetMaxProductionCount   : BOOL;
    bResetTotalProductionCount : BOOL;

    nMaxProductionCount   : DINT;
    nTotalProductionCount : DINT;

    stProductionDataHMI          : ST_ProductionData_HMI;
    fbFIFO                       : FB_FIFO_ULINT_Array;
    a_fbProductionDataAlarms     : ARRAY[1..PRODUCTION_DATA_ALARM_COUNT] OF FB_TcAlarm;
    fTemp                        : LREAL;
    bInitialized                 : BOOL;
    initialize                   : INT;
    fLastProductionRate_Setpoint : LREAL;
END_VAR

PROPERTY CurrentShiftAcceptableProduction : DINT
GET
END_GET
SET
END_SET
END_PROPERTY

PROPERTY CurrentShiftProductionCount : DINT
GET
CurrentShiftProductionCount := nCurrentShiftProductionCount;
END_GET
END_PROPERTY

PROPERTY CurrentShiftTarget : DINT
GET
CurrentShiftTarget := nCurrentShiftTarget;
END_GET
END_PROPERTY

PROPERTY CurrentShiftTime : TIME
GET
CurrentShiftTime := tCurrentShiftTime;
END_GET
END_PROPERTY

PROPERTY CurrentShiftWarningProduction : DINT
GET
END_GET
SET
END_SET
END_PROPERTY

METHOD HMICommunication : BOOL
VAR_INPUT
END_VAR
//Production Data================================================================================================================================================

//Process HMI requests
IF stProductionDataHMI.bIncomingHMIRequest AND NOT stProductionDataHMI.bHMICommandConfirmation
    THEN //If a request has been issued by the HMI, and a previous request has not just E_SequenceState.Finished being processed
    IF stProductionDataHMI.bShiftProductionTargetHMISetRequest THEN
        nShiftProductionTarget                      := stProductionDataHMI.nShiftProductionTargetHMISetValue;
        stProductionDataHMI.bHMICommandConfirmation := TRUE; //Confirm that the request has been processed
    END_IF

    IF stProductionDataHMI.bWarningMarginHMISetRequest THEN
        fWarningMargin                              := stProductionDataHMI.fWarningMarginHMISetValue;
        stProductionDataHMI.bHMICommandConfirmation := TRUE; //Confirm that the request has been processed
    END_IF

    IF stProductionDataHMI.bShiftLengthHMISetRequest THEN
        tShiftLength                                := stProductionDataHMI.tShiftLengthHMISetValue;
        stProductionDataHMI.bHMICommandConfirmation := TRUE; //Confirm that the request has been processed
    END_IF

    IF stProductionDataHMI.bProductionRateHMISetRequest THEN
        fProductionRate_Setpoint                    := stProductionDataHMI.fProductionRateHMISetValue;
        stProductionDataHMI.bHMICommandConfirmation := TRUE; //Confirm that the request has been processed
    END_IF
END_IF

//Update HMI Status Info
stProductionDataHMI.tShiftLength                      := tShiftLength;
stProductionDataHMI.nShiftProductionTarget            := nShiftProductionTarget;
stProductionDataHMI.nCurrentShiftProductionCount      := nCurrentShiftProductionCount;
stProductionDataHMI.nCurrentShiftTarget               := nCurrentShiftTarget;
stProductionDataHMI.nCurrentAcceptableProductionCount := nCurrentAcceptableProductionCount;
stProductionDataHMI.nCurrentWarningProductionCount    := nCurrentWarningProductionCount;
stProductionDataHMI.tCurrentShiftTime                 := tCurrentShiftTime;
stProductionDataHMI.tRemainingShiftTime               := tRemainingShiftTime;
stProductionDataHMI.fProductionRate_Setpoint          := F_LREAL_RoundToPlace(fProductionRate_Setpoint, 1);
stProductionDataHMI.fProductionRate_Actual            := F_LREAL_RoundToPlace(fProductionRate_Actual, 1);
stProductionDataHMI.fProductionRate_Required          := F_LREAL_RoundToPlace(fProductionRate_Required, 1);
END_METHOD

METHOD initialize : BOOL
VAR_INPUT
END_VAR
END_METHOD

METHOD Monitor : BOOL
VAR_INPUT
END_VAR
IF NOT bInitialized THEN
    initialize();
    bInitialized := TRUE;
END_IF

fbFIFO(a_FIFO := a_nLastProductTimestamps);

fbShiftTimer(IN := NOT bShiftComplete, PT := tShiftLength, Q => bShiftComplete, ET => tCurrentShiftTime);
tRemainingShiftTime := tShiftLength - tCurrentShiftTime;

IF TIME_TO_DINT(tRemainingShiftTime) > 0 THEN
    fProductionRate_Required :=
        DINT_TO_LREAL(nShiftProductionTarget - nCurrentShiftProductionCount) / (TIME_TO_LREAL(tRemainingShiftTime) / 1000 / 60);

    nCurrentAcceptableProductionCount := nCurrentShiftTarget;

    nCurrentWarningProductionCount :=
        nShiftProductionTarget
            - (LREAL_TO_DINT((fProductionRate_Actual * (1 + fWarningMargin / 100)) * (TIME_TO_LREAL(tRemainingShiftTime) / 1000 / 60)));

    IF nCurrentWarningProductionCount < 0 THEN
        nCurrentWarningProductionCount := 0;
    END_IF
END_IF

fbProductComplete_RT(CLK := bProductComplete);

IF fbProductComplete_RT.Q THEN
    nCurrentShiftProductionCount := nCurrentShiftProductionCount + 1;
    nTotalProductionCount        := nTotalProductionCount + 1;

    IF nCurrentShiftProductionCount > nMaxProductionCount THEN
        nMaxProductionCount := nCurrentShiftProductionCount;
    END_IF

    fbFIFO.AddEntry(nEntry := F_GetSystemTime());
END_IF

IF (fbFIFO.EntryCount > nRateAveragingCount) THEN
    fbFIFO.RemoveEntry();
END_IF

fTemp := (TIME_TO_LREAL(ULINT_TO_TIME(fbFIFO.LastInValue - fbFIFO.NextOutValue)) / 10000 / 1000 / 60);

IF fTemp > 0 AND fbFIFO.EntryCount > 1 THEN
    fProductionRate_Actual := F_LREAL_RoundToPlace(DINT_TO_LREAL(fbFIFO.EntryCount - 1) / fTemp, 2);
END_IF

IF TIME_TO_DINT(tShiftLength) > 0 THEN
    nCurrentShiftTarget := LREAL_TO_DINT((TIME_TO_LREAL(tCurrentShiftTime) / TIME_TO_LREAL(tShiftLength)) * DINT_TO_LREAL(nShiftProductionTarget));
END_IF

IF bShiftComplete THEN
    nCurrentShiftProductionCount := 0;
END_IF

IF bResetMaxProductionCount THEN
    nMaxProductionCount := nCurrentShiftProductionCount;
END_IF

IF bResetTotalProductionCount THEN
    nTotalProductionCount := 0;
END_IF

IF fProductionRate_Setpoint <> fLastTargetProductionRate THEN
    bNewProductionRate := TRUE;
ELSE
    bNewProductionRate := FALSE;
END_IF

fLastTargetProductionRate := fProductionRate_Setpoint;
END_METHOD

PROPERTY NewProductionRate : BOOL
GET
NewProductionRate := bNewProductionRate;
END_GET
END_PROPERTY

PROPERTY ProductComplete : BOOL
GET
ProductComplete := bProductComplete;
END_GET
SET
bProductComplete := ProductComplete;
END_SET
END_PROPERTY

PROPERTY ProductionRate_Actual : LREAL
GET
ProductionRate_Actual := fProductionRate_Actual;
END_GET
END_PROPERTY

PROPERTY ProductionRate_Required : LREAL
GET
ProductionRate_Required := fProductionRate_Required;
END_GET
SET
fProductionRate_Required := ProductionRate_Required;
END_SET
END_PROPERTY

PROPERTY ProductionRate_Setpoint : LREAL
GET
ProductionRate_Setpoint := fProductionRate_Setpoint;
END_GET
SET
fProductionRate_Setpoint := ProductionRate_Setpoint;
END_SET
END_PROPERTY

PROPERTY RateAveragingCount : DINT
GET
RateAveragingCount := nRateAveragingCount;
END_GET
SET
nRateAveragingCount := RateAveragingCount;
END_SET
END_PROPERTY

PROPERTY RemainingShiftTime : TIME
GET
END_GET
SET
END_SET
END_PROPERTY

PROPERTY ShiftComplete : BOOL
GET
ShiftComplete := bShiftComplete;
END_GET
END_PROPERTY

PROPERTY ShiftLength : TIME
GET
ShiftLength := tShiftLength;
END_GET
SET
tShiftLength := ShiftLength;
END_SET
END_PROPERTY

PROPERTY ShiftProductionTarget : DINT
GET
ShiftProductionTarget := nShiftProductionTarget;
END_GET
SET
nShiftProductionTarget := ShiftProductionTarget;
END_SET
END_PROPERTY

PROPERTY WarningMargin : LREAL
GET
WarningMargin := fWarningMargin;
END_GET
SET
fWarningMargin := WarningMargin;
END_SET
END_PROPERTY

END_FUNCTION_BLOCK

// ---- Application/02_MachineModules/FB_TestMachine.TcPOU
FUNCTION_BLOCK FB_TestMachine EXTENDS FB_PMLModuleBase
VAR
    //Define the Sub modules here for this module.  Also set the Interfaces in the initialize method.
    //fbSubModule1				: FB_ApplicationModule_TEMPLATE;		// Sub module instantiation
    //fbSubModule2				: FB_ApplicationModule_TEMPLATE;		// Sub module instantiation

    fbEquipmentModule1 : FB_TestEquipment := (ModuleName := 'Equipment Module 1');
	fbEquipmentModule2 : FB_TestEquipment := (ModuleName := 'Equipment Module 2');
	fbEquipmentModule3 : FB_TestEquipment := (ModuleName := 'Equipment Module 3');

    //temporary array of module base interfaces to be copied over to the base class itfPackMLBase variable
    a_itfPackMLBase_init : ARRAY[1..MAX_NO_OF_SUBMODULES] OF ITF_PMLModuleBase := [fbEquipmentModule1, fbEquipmentModule2, fbEquipmentModule3] (*, fbSubModule2,*) ;

    //Define the components here for this module. (If any) Also set the Interfaces in the initialize method.
    (*fbComponent1				: FB_ComponentBase (Extension):= (Name := 'Test Component 1');
	*)
    (*fbComponent2				: FB_ComponentBase (Extension):= (Name := 'Test Component 2');
	*)

    //temporary array of module base interfaces to be copied over to the base class a_itfPackMLBase variable
    a_ITF_Components_init : ARRAY[1..GVL_PML_Base.MAX_NO_OF_COMPONENTS] OF ITF_ComponentBase := [ (*fbComponent1,fbComponent2*) ];

    // Other machine specific variables here
END_VAR

//*********************************************************
// Code implementation only in Execute() method for consistency with templates
//*********************************************************

// 
// Cyclic Code
METHOD CyclicLogic
VAR
    i : UDINT; //Generic iteration value
END_VAR
FOR i := 1 TO 5 DO
    a_sModeNames[i] := F_UnitModeToString(i);
	
END_FOR

// Main loop of the parent module
SUPER^.CyclicLogic();
END_METHOD

METHOD Initialize
VAR
    i : UDINT; //Generic iteration value
END_VAR
// Define the interfaces to the different subunits (Must take place before SUPER^.initialize call)
FOR i := 1 TO MAX_NO_OF_SUBMODULES DO
    a_ITF_PackMLBase[i] := a_itfPackMLBase_init[i];
END_FOR

FOR i := 1 TO MAX_NO_OF_COMPONENTS DO
    a_ITF_Components[i] := a_ITF_Components_init[i];
END_FOR

// Init of the parent class object (Must be called AFTER most local init code, since the sub module interface array assignments should be made here, and then operated on within the module base init
SUPER^.Initialize();
END_METHOD

END_FUNCTION_BLOCK

// ---- Application/03_EquipmentModules/FB_TestEquipment.TcPOU
FUNCTION_BLOCK FB_TestEquipment EXTENDS FB_PMLModuleBase
VAR
    //Define the Sub modules here for this module.  Also set the Interfaces in the initialize method.

    //temporary array of module base interfaces to be copied over to the base class itfPackMLBase variable
    a_itfPackMLBase_init : ARRAY[1..MAX_NO_OF_SUBMODULES] OF ITF_PMLModuleBase := [];

    //Define the components here for this module. (If any) Also set the Interfaces in the initialize method.
    (*fbComponent1				: FB_ComponentBase (Extension):= (Name := 'Test Component 1');
	*)
    (*fbComponent2				: FB_ComponentBase (Extension):= (Name := 'Test Component 2');
	*)
    //temporary array of module base interfaces to be copied over to the base class a_itfPackMLBase variable

    a_ITF_Components_init : ARRAY[1..GVL_PML_Base.MAX_NO_OF_COMPONENTS] OF ITF_ComponentBase := [];

    // Other machine specific variables here
END_VAR

//*********************************************************
// Code implementation only in Execute() method for consistency with templates
//*********************************************************

// 
// Cyclic Code
METHOD CyclicLogic
VAR
    i : UDINT; //Generic iteration value
END_VAR
FOR i := 1 TO 5 DO
    a_sModeNames[i] := F_UnitModeToString(i);
	
END_FOR



// Main loop of the parent module
SUPER^.CyclicLogic();
END_METHOD

METHOD Initialize
VAR
    i : UDINT; //Generic iteration value
END_VAR
// Define the interfaces to the different subunits (Must take place before SUPER^.initialize call)
FOR i := 1 TO MAX_NO_OF_SUBMODULES DO
    a_ITF_PackMLBase[i] := a_itfPackMLBase_init[i];
END_FOR

FOR i := 1 TO MAX_NO_OF_COMPONENTS DO
    a_ITF_Components[i] := a_ITF_Components_init[i];
END_FOR

// Init of the parent class object (Must be called AFTER most local init code, since the sub module interface array assignments should be made here, and then operated on within the module base init
SUPER^.Initialize();
END_METHOD

END_FUNCTION_BLOCK

// ---- Application/04_Components/01_Cylinder_Example/FB_CylinderBase.TcPOU
FUNCTION_BLOCK ABSTRACT FB_CylinderBase EXTENDS FB_ComponentBase IMPLEMENTS ITF_CylinderBase //Abstract (non-instantiable) base definition from which numerous varieties of Cylinders may be derived through function block extension.
VAR_INPUT
END_VAR
VAR_OUTPUT
END_VAR
VAR CONSTANT
    //Constant declarations
    CYLINDER_BASE_ALARM_COUNT : UDINT := 16;
END_VAR
VAR
    //ITF_Cylinder internal property variables
    tExtendTime    : TIME  := T#3S; //Approximate expected time for the cylinder to complete an extension cycle
    tRetractTime   : TIME  := T#3S; //Approximate expected time for the cylinder to complete a retraction cycle
    fTimeoutFactor : LREAL := 1.5;  //Multiplicative factor that determines error timeout threshold based on the expected cycle time
    bExtended      : BOOL;          //Status bit for the position of the cylinder
    bRetracted     : BOOL;          //Status bit for the position of the cylinder
    bExtending     : BOOL;          //Cylinder is currently extending
    bRetracting    : BOOL;          //Cylinder is currently retracting
    bExtendOutput  : BOOL;          //Cylinder "extend" output is currently active
    bRetractOutput : BOOL;          //Cylinder "retract" output is currently active

    //Alarming
    a_fbCylinderBaseAlarms : ARRAY[1..CYLINDER_BASE_ALARM_COUNT] OF FB_TcAlarm;

    //HMI monitoring and control structure
    stCylinderBaseHMI : ST_CylinderBase_HMI;

    //Internal Variables
    fbExtensionTimeout_TON  : Tc2_Standard.TON; //Timer for monitoring extension timeouts
    tExtensionTimeout       : TIME;             //Extension timeout threshold calculated from expected ExtendTime and TimeoutFactor
    fbRetractionTimeout_TON : Tc2_Standard.TON; //Timer for monitoring retraction timeouts
    tRetractionTimeout      : TIME;             //Retraction timeout threshold calculated from expected RetractTime and TimeoutFactor
    bExtendRequest          : BOOL;             //Extension request received
    bRetractRequest         : BOOL;             //Retraction request received
    bExtendCommand          : BOOL;             //Direct command to be sent to outputs
    bRetractCommand         : BOOL;             //Direct command to be sent to outputs
    bExtendedFeedback       : BOOL;             //Direct feedback value from inputs
    bRetractedFeedback      : BOOL;             //Direct feedback value from inputs
    bIncomingRequest        : BOOL;             //New external request has been made

    //Simulation variables
    fbSimExtend_TON    : Tc2_Standard.TON;
    fbSimRetract_TON   : Tc2_Standard.TON;
    bSimExtendCommand  : BOOL;
    bSimRetractCommand : BOOL;
END_VAR

METHOD AllowHMIControl : BOOL
VAR_INPUT
END_VAR
SUPER^.AllowHMIControl();

stCylinderBaseHMI.bHMIControlAvailable := TRUE;
END_METHOD

METHOD BlockHMIControl : BOOL
VAR_INPUT
END_VAR
SUPER^.BlockHMIControl();

stCylinderBaseHMI.bHMIControlAvailable := FALSE;
END_METHOD

//{attribute 'call_after_online_change_slot' := '<slot>'}
METHOD CreateEvents : BOOL
VAR_INPUT
END_VAR
SUPER^.CreateEvents();

F_CreateAllEventsInClass(p_aAlarms  := a_fbCylinderBaseAlarms,
                         nClassSize := SIZEOF(TC_EVENTS.CylinderBase),
                         pInitEvent := ADR(TC_EVENTS.CylinderBase.InitReferenceEvent),
                         sPrefix    := sName);
END_METHOD

METHOD ErrorOperation : BOOL
VAR_INPUT
END_VAR
bExtendCommand  := FALSE;
bRetractCommand := FALSE;
END_METHOD

METHOD Extend : BOOL
bExtendRequest   := TRUE;
bRetractRequest  := FALSE;
bIncomingRequest := TRUE;
END_METHOD

{attribute 'monitoring' := 'variable'}
PROPERTY Extended : BOOL //Status bit for the position of the cylinder
GET
Extended := bExtended;
END_GET
END_PROPERTY

PROPERTY Extending : BOOL
GET
Extending := bExtending;
END_GET
END_PROPERTY

PROPERTY ExtendOutput : BOOL
GET
ExtendOutput := bExtendOutput;
END_GET
END_PROPERTY

PROPERTY ExtendTime : TIME //Approximate expected time for the cylinder to complete an extension cycle
GET
ExtendTime := tExtendTime;
END_GET
SET
tExtendTime := ExtendTime;
END_SET
END_PROPERTY

METHOD GenerateFeedback : BOOL
VAR_INPUT
    bExtend  : BOOL;
    bRetract : BOOL;
END_VAR
VAR_OUTPUT
    bExtended_Generated  : BOOL;
    bRetracted_Generated : BOOL;
END_VAR
VAR_INST
    bLastExtend    : BOOL;
    bLastRetract   : BOOL;
    bExtendedTemp  : BOOL;
    bRetractedTemp : BOOL;
END_VAR
IF bExtend AND NOT bLastExtend THEN //Whenever a new extend request comes in, check to see if we are still currently timing a retract action
    IF fbSimRetract_TON.IN AND NOT bRetracted_Generated
        THEN //If a retract action is still in progress, appropriately scale the extend time to account for the distance traveled during the in-process retraction
        fbSimExtend_TON.PT := tExtendTime
                                  * (TIME_TO_UDINT(fbSimRetract_TON.ET) / TIME_TO_UDINT(tRetractTime)
                                  ); //partial extend time = (full distance extend time) * (proportional distance covered during retraction)

        fbSimRetract_TON.IN := FALSE; //Disable retract timer
    ELSIF NOT fbSimExtend_TON.IN THEN
        fbSimExtend_TON.PT := tExtendTime; //If no retraction was active, assume we are currently at fully retracted position, or this is the first command the cylinder has received, so initialize to full extend time
    END_IF

    bRetractedTemp     := FALSE;
    fbSimExtend_TON.IN := TRUE;          //Activate the extension timer
ELSIF bRetract AND NOT bLastRetract THEN //Same as above, but reversed
    IF fbSimExtend_TON.IN AND NOT bExtended_Generated THEN
        fbSimRetract_TON.PT := tRetractTime * (TIME_TO_UDINT(fbSimExtend_TON.ET) / TIME_TO_UDINT(tRetractTime));
        fbSimExtend_TON.IN  := FALSE;
    ELSIF NOT fbSimRetract_TON.IN THEN
        fbSimRetract_TON.PT := tRetractTime;
    END_IF

    bExtendedTemp       := FALSE;
    fbSimRetract_TON.IN := TRUE;
END_IF

bLastExtend  := bExtend;
bLastRetract := bRetract;

IF fbSimExtend_TON.Q THEN //Whenever the extend timer completes, set status to extended and turn off the timer
    bExtendedTemp      := TRUE;
    fbSimExtend_TON.IN := FALSE;
END_IF

IF fbSimRetract_TON.Q THEN //Whenever the retract timer completes, set status to retracted and turn off the timer
    bRetractedTemp      := TRUE;
    fbSimRetract_TON.IN := FALSE;
END_IF

bExtended_Generated  := bExtendedTemp;
bRetracted_Generated := bRetractedTemp;
END_METHOD

METHOD HMICommunication : BOOL
SUPER^.HMICommunication(); //Call the base method

//Process HMI requests
IF stCylinderBaseHMI.bIncomingHMIRequest AND NOT stCylinderBaseHMI.bHMICommandConfirmation
    THEN //If a request has been issued by the HMI, and a previous request has not just finished being processed
    IF stCylinderBaseHMI.bHMIControlAvailable
        THEN //If the current conditions permit HMI control (Should be determined by the extended application components)
        IF stCylinderBaseHMI.bExtendHMIRequest
            THEN //Execute the active requests
            Extend();
            stCylinderBaseHMI.bHMICommandConfirmation := TRUE; //Confirm that the request has been processed
        END_IF

        IF stCylinderBaseHMI.bRetractHMIRequest THEN
            Retract();
            stCylinderBaseHMI.bHMICommandConfirmation := TRUE; //Confirm that the request has been processed
        END_IF

        IF stCylinderBaseHMI.bIdleHMIRequest THEN
            Idle();
            stCylinderBaseHMI.bHMICommandConfirmation := TRUE; //Confirm that the request has been processed
        END_IF

        IF stCylinderBaseHMI.bExtendTimeHMISetRequest THEN
            ExtendTime                                := stCylinderBaseHMI.tExtendTimeHMISetValue;
            stCylinderBaseHMI.bHMICommandConfirmation := TRUE; //Confirm that the request has been processed
        END_IF

        IF stCylinderBaseHMI.bRetractTimeHMISetRequest THEN
            RetractTime                               := stCylinderBaseHMI.tRetractTimeHMISetValue;
            stCylinderBaseHMI.bHMICommandConfirmation := TRUE; //Confirm that the request has been processed
        END_IF

        IF stCylinderBaseHMI.bTimeoutFactorHMISetRequest THEN
            TimeoutFactor                             := stCylinderBaseHMI.fTimeoutFactorHMISetValue;
            stCylinderBaseHMI.bHMICommandConfirmation := TRUE; //Confirm that the request has been processed
        END_IF
    END_IF
END_IF

//Update HMI status info
stCylinderBaseHMI.tExtendTime     := tExtendTime;
stCylinderBaseHMI.tRetractTime    := tRetractTime;
stCylinderBaseHMI.fTimeoutFactor  := fTimeoutFactor;
stCylinderBaseHMI.bExtended       := bExtended;
stCylinderBaseHMI.bExtending      := bExtending;
stCylinderBaseHMI.bRetracted      := bRetracted;
stCylinderBaseHMI.bRetracting     := bRetracting;
stCylinderBaseHMI.bExtendCommand  := bExtendCommand OR bSimExtendCommand;
stCylinderBaseHMI.bRetractCommand := bRetractCommand OR bSimRetractCommand;
END_METHOD

METHOD Idle : BOOL
bExtendRequest   := FALSE;
bRetractRequest  := FALSE;
bIncomingRequest := TRUE;

bExtendCommand  := FALSE;
bRetractCommand := FALSE;
END_METHOD

METHOD initialize : BOOL
VAR_INPUT
END_VAR

VAR
    sTemp : STRING;
END_VAR
SUPER^.initialize();
END_METHOD

METHOD Monitoring : BOOL
VAR_INPUT
END_VAR
tExtensionTimeout  := LREAL_TO_TIME(TIME_TO_LREAL(tExtendTime) * fTimeoutFactor);
tRetractionTimeout := LREAL_TO_TIME(TIME_TO_LREAL(tRetractTime) * fTimeoutFactor);

fbExtensionTimeout_TON(IN := bExtending,
                       PT := tExtensionTimeout); //Timer for monitoring extension timeout, PT = Extension time multiplied by the timeout factor

fbRetractionTimeout_TON(IN := bRetracting,
                        PT := tRetractionTimeout); //Timer for monitoring retraction timeout, PT = Retraction time multiplied by the timeout factor

IF NOT bError THEN

    //Simultaneous extend and retract commands throw an invalid command error
    IF (bExtending AND bRetracting) OR (bExtendRequest AND bRetractRequest) OR (bExtendCommand AND bRetractCommand) THEN
        IF NOT a_fbCylinderBaseAlarms[E_CylinderBase.InvalidCommand].bRaised THEN
            RaiseAlarm(fbAlarm := a_fbCylinderBaseAlarms[E_CylinderBase.InvalidCommand]);
        END_IF
    ELSIF a_fbCylinderBaseAlarms[E_CylinderBase.InvalidCommand].bRaised THEN
        a_fbCylinderBaseAlarms[E_CylinderBase.InvalidCommand].Clear(0, 0);
    END_IF

    //If both extended and retracted feedback are true at any point, throw an invalid position error
    IF bExtended AND bRetracted THEN
        IF NOT a_fbCylinderBaseAlarms[E_CylinderBase.InvalidPositionStatus].bRaised THEN
            RaiseAlarm(fbAlarm := a_fbCylinderBaseAlarms[E_CylinderBase.InvalidPositionStatus]);
        END_IF
    ELSIF a_fbCylinderBaseAlarms[E_CylinderBase.InvalidPositionStatus].bRaised THEN
        a_fbCylinderBaseAlarms[E_CylinderBase.InvalidPositionStatus].Clear(0, 0);
    END_IF

    //If the cylinder takes longer than expected to extend, throw a timeout error
    IF fbExtensionTimeout_TON.Q THEN
        IF NOT a_fbCylinderBaseAlarms[E_CylinderBase.ExtendTimeout].bRaised THEN
            RaiseAlarmWithStrings(fbAlarm := a_fbCylinderBaseAlarms[E_CylinderBase.ExtendTimeout], TIME_TO_STRING(tExtensionTimeout), '');
        END_IF
    ELSIF a_fbCylinderBaseAlarms[E_CylinderBase.ExtendTimeout].bRaised THEN
        a_fbCylinderBaseAlarms[E_CylinderBase.ExtendTimeout].Clear(0, 0);
    END_IF

    //If the cylinder takes longer than expected to retract, throw a timeout error
    IF fbRetractionTimeout_TON.Q THEN
        IF NOT a_fbCylinderBaseAlarms[E_CylinderBase.RetractTimeout].bRaised THEN
            RaiseAlarmWithStrings(fbAlarm := a_fbCylinderBaseAlarms[E_CylinderBase.RetractTimeout], TIME_TO_STRING(tRetractionTimeout), '');
        END_IF
    ELSIF a_fbCylinderBaseAlarms[E_CylinderBase.RetractTimeout].bRaised THEN
        a_fbCylinderBaseAlarms[E_CylinderBase.RetractTimeout].Clear(0, 0);
    END_IF
END_IF

//If cylinder is in motion toward a position, but it has not yet been reached, set busy bit
IF (bExtending) OR (bRetracting) THEN
    bActive := TRUE;
ELSE
    bActive := FALSE;
END_IF

IF bSimExtendCommand OR bExtendCommand THEN
    bExtendOutput := TRUE;
ELSE
    bExtendOutput := FALSE;
END_IF

IF bSimRetractCommand OR bRetractCommand THEN
    bRetractOutput := TRUE;
ELSE
    bRetractOutput := FALSE;
END_IF

IF bRetractOutput AND NOT bRetracted THEN
    bRetracting := TRUE;
ELSE
    bRetracting := FALSE;
END_IF

IF bExtendOutput AND NOT bExtended THEN
    bExtending := TRUE;
ELSE
    bExtending := FALSE;
END_IF

bReady := bEnabled AND NOT bError;

eCurrentAlarmSeverity := F_GetMaxSeverityRaised(a_fbAlarms := a_fbCylinderBaseAlarms, eCurrentSeverity := eCurrentAlarmSeverity);

SUPER^.Monitoring();
END_METHOD

METHOD Reset : BOOL
SUPER^.Reset();
bError := FALSE;

fbSimExtend_TON.IN  := FALSE;
fbSimRetract_TON.IN := FALSE;

bExtendCommand     := FALSE;
bRetractCommand    := FALSE;
bSimExtendCommand  := FALSE;
bSimRetractCommand := FALSE;
END_METHOD

METHOD Retract : UDINT
bRetractRequest  := TRUE;
bExtendRequest   := FALSE;
bIncomingRequest := TRUE;
END_METHOD

{attribute 'monitoring' := 'variable'}
PROPERTY Retracted : BOOL //Status bit for the position of the cylinder
GET
Retracted := bRetracted;
END_GET
END_PROPERTY

PROPERTY Retracting : BOOL
GET
Retracting := bRetracting;
END_GET
END_PROPERTY

PROPERTY RetractOutput : BOOL
GET
RetractOutput := bRetractOutput;
END_GET
END_PROPERTY

PROPERTY RetractTime : TIME
GET
RetractTime := tRetractTime;
END_GET
SET
tRetractTime := RetractTime;
END_SET
END_PROPERTY

METHOD SimulateOperation : BOOL
VAR_INPUT
END_VAR
bExtendCommand  := FALSE; //Hardware commands should be disabled during simulation mode
bRetractCommand := FALSE; //Hardware commands should be disabled during simulation mode

IF bEnabled THEN
    IF bIncomingRequest THEN
        bSimExtendCommand  := bExtendRequest;
        bSimRetractCommand := bRetractRequest;
        bIncomingRequest   := FALSE;
    END_IF

    fbSimExtend_TON();  //Call timer FB
    fbSimRetract_TON(); //Call timer FB

    GenerateFeedback(bExtend              := bSimExtendCommand,
                     bRetract             := bSimRetractCommand,
                     bExtended_Generated  => bExtended,
                     bRetracted_Generated => bRetracted);
ELSE
    bIncomingRequest    := FALSE;
    fbSimExtend_TON.IN  := FALSE;
    fbSimRetract_TON.IN := FALSE;
END_IF
END_METHOD

METHOD StandardOperation : BOOL
VAR_INPUT
END_VAR
IF bEnabled THEN
    IF bIncomingRequest THEN
        bExtendCommand   := bExtendRequest;
        bRetractCommand  := bRetractRequest;
        bIncomingRequest := FALSE;
    END_IF

    bExtended  := bExtendedFeedback;
    bRetracted := bRetractedFeedback;
ELSE
    bIncomingRequest := FALSE;
END_IF
END_METHOD

PROPERTY TimeoutFactor : LREAL //Multiplicative factor that determines error timeout threshold based on the expected time
GET
TimeoutFactor := fTimeoutFactor;
END_GET
SET
fTimeoutFactor := TimeoutFactor;
END_SET
END_PROPERTY

END_FUNCTION_BLOCK

// ---- Application/MAIN.TcPOU
PROGRAM MAIN
VAR
    fbMainModuleHMIConnection : FB_MainModule_HMI_Connection;

    // Define the top level Machine as defined in the Application/01_MachineModules folder here
    fbMyMachine : FB_TestMachine := (MasterDataStructure_Adder := fbMainModuleHMIConnection.DataStructure_Adder, LogStateChanges := TRUE,
                                     ModuleID := 1, ModuleName := 'My Machine Module');

    bInitialized : BOOL;
END_VAR

CyclicLogic();

METHOD CyclicLogic : BOOL
VAR_INPUT
END_VAR
IF NOT bInitialized THEN
    Initialize();
    bInitialized := TRUE;
END_IF

fbMainModuleHMIConnection.CyclicLogic();

//The Top level machine CyclicLogic call should be made here, all sub modules should be called from within their respective parent CyclicLogic methods
fbMyMachine.CyclicLogic();

// Add other Main CyclicLogic here
END_METHOD

METHOD Initialize : BOOL
VAR_INPUT
END_VAR
//Top level machine initialization should happen here, in the main initialization method. Each subsequent "layer" of modules will be named within their respective "parent" intialize method
fbMainModuleHMIConnection.MainModule := fbMyMachine;
END_METHOD

END_PROGRAM
